TEXTLIST TL_EventServerity
  0 = 'Verbose'
  1 = 'Info'
  2 = 'Warning'
  3 = 'Error'
  4 = 'Critical'
   = ''
END_TEXTLIST

(* stored: Version 1.1.0.1, ProductVersion 3.1.4024.9
   TextList TL_EventServerity: Id {1f48cbbf-0860-4d0b-9c2a-70478ac00e1c} *)
